(* PLC project Unnamed, Unknown Unnamed 1 *)
(* stored: creationDateTime 2024-01-09T16:45:07, modificationDateTime 2024-01-23T14:31:54 *)

FUNCTION_BLOCK Reals_MultiplyByParameter
  VAR_INPUT
    u : REAL;
    k : REAL;
  END_VAR
  VAR_OUTPUT
    y : REAL;
  END_VAR

						y := k * u;
					
END_FUNCTION_BLOCK

PROGRAM Custom02
  VAR_INPUT
    ymax : REAL;
    ymax1 : REAL;
  END_VAR
  VAR_OUTPUT
    y : REAL;
    y1 : REAL;
  END_VAR
  VAR
    gain : Reals_MultiplyByParameter;
    gain1 : Reals_MultiplyByParameter;
    r1 : REAL := 1.0;
  END_VAR

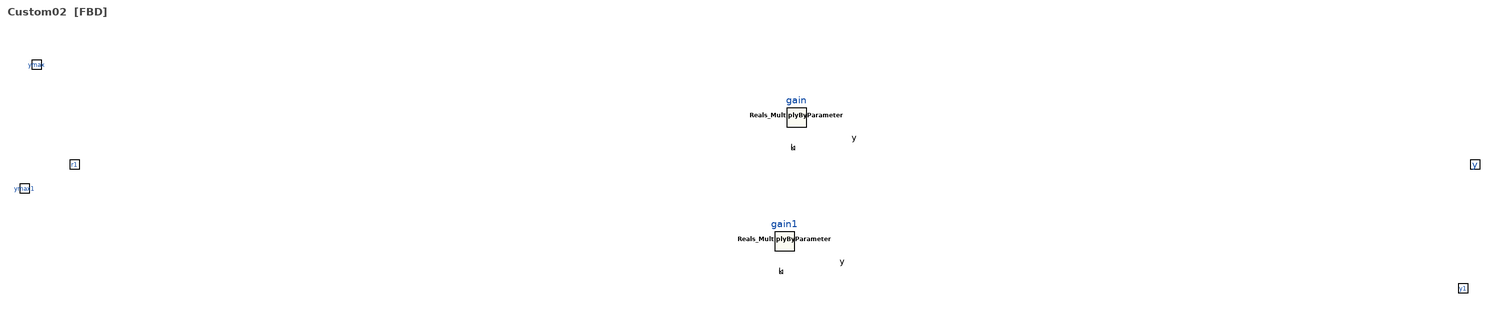
(* FBD diagram, written out as Structured Text *)
gain(u := ymax, k := r1);
y := gain.y;
gain1(u := ymax1, k := r1);
y1 := gain1.y;
END_PROGRAM

CONFIGURATION config
  RESOURCE resource1 ON PLC
    TASK task0(INTERVAL := T#20ms, PRIORITY := 0);
    PROGRAM instance0 WITH task0 : Custom02;
  END_RESOURCE
END_CONFIGURATION
